FUNCTION F_TB_Tx_BCC : STRING
VAR_INPUT
	txStr: STRING;
END_VAR
VAR
	i, len1: INT;
	bArr: ARRAY[0..255] OF BYTE;
	b1: BYTE;
END_VAR

// SMC HEBC002-WA10
len1 := LEN(STR:=txStr);
len1 := len1 - 1;
bArr := MAXSTRING_TO_BYTEARR(txStr);
FOR i := 0 TO len1 DO
	b1 := b1 XOR bArr[i];
END_FOR
F_TB_Tx_BCC := F_toCHR(b1);

END_FUNCTION

(* stored: Version 1.1.0.1, ProductVersion 3.1.4024.12
   POU F_TB_Tx_BCC: Id {ebb9db4f-bc1e-4c29-af55-f290b332d2a1}, SpecialFunc None *)
